RoboDK station: Robotska celija zadnja verzija.rdk

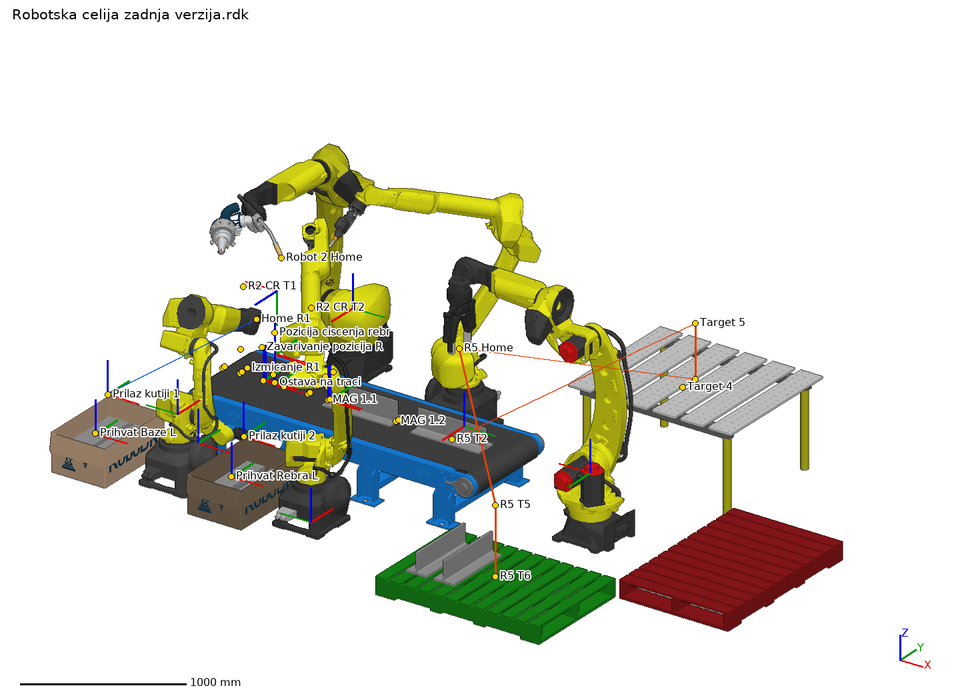
[picture v0: the station drawn from its stored meshes, robots at their saved joint values, targets as dots, program paths as lines]
Station Robotska celija zadnja verzija (saved by RoboDK 5.3.0). Poses are relative to the parent item; angles as X-Y-Z fixed-axis rotations.
  - program MAIN R12345 (8 instructions, listed below)
  - frame Frame Conveyor at (1000, 1000, 0) mm
    - robot Conveyor Belt Wide (2m): 1 axes
        modified DH rows (alpha deg, a mm, theta deg, d mm): 0, 0, 0, 0 linear
        base shift (0, 0, 0) mm, rotated rx 0 ry 90 rz 0 deg
        joint limits [-900000] to [900000]; home [0]; saved at [0]
  - frame R1 Frame at (1200, 500, 450) mm, rotated rx 0 ry 0 rz 90 deg
    - robot Fanuc M-10iD/16S: 6 axes
        modified DH rows (alpha deg, a mm, theta deg, d mm): 0, 0, 0, 450; -90, 75, -90, 0; 0, 440, 0, 0; -90, 195, 180, 555; 90, 0, 0, 0; -90, 0, 90, 90
        base shift (0, 0, -450) mm
        joint limits [-185, -90, -200, -190, -180, -450] to [185, 145, 200, 190, 180, 450]; home [0, 0, 0, 0, 0, 0]; saved at [0, 0, -25, 0, 0, 0]
      - tool OnRobot MG10 Magnetic Gripper, TCP at (0, 0, 93) mm, size 71 x 74.9 x 91.4 mm
  - object Kutija - baze at (500, 170, 0) mm, size 424.8 x 637.2 x 266.3 mm, geometry from Box-24x16in-Open.sld
    - object Baza L at (110, 310, 0) mm, rotated rx 0 ry 0 rz 90 deg, size 500 x 150 x 16 mm, geometry from Baza.step
      - object Baza at (0, 0, 16) mm, size 500 x 150 x 16 mm, geometry from Baza.step
        - object Baza at (0, 0, 16) mm, size 500 x 150 x 16 mm, geometry from Baza.step
          - object Baza at (0, 0, 16) mm, size 500 x 150 x 16 mm, geometry from Baza.step
            - object Baza at (0, 0, 16) mm, size 500 x 150 x 16 mm, geometry from Baza.step
              - object Baza at (0, 0, 16) mm, size 500 x 150 x 16 mm, geometry from Baza.step
    - object Baza D at (290, 310, 0) mm, rotated rx 0 ry 0 rz 90 deg, size 500 x 150 x 16 mm, geometry from Baza.step
      - object Baza at (0, 0, 16) mm, size 500 x 150 x 16 mm, geometry from Baza.step
        - object Baza at (0, 0, 16) mm, size 500 x 150 x 16 mm, geometry from Baza.step
          - object Baza at (0, 0, 16) mm, size 500 x 150 x 16 mm, geometry from Baza.step
            - object Baza at (0, 0, 16) mm, size 500 x 150 x 16 mm, geometry from Baza.step
              - object Baza at (0, 0, 16) mm, size 500 x 150 x 16 mm, geometry from Baza.step
                - object Baza at (0, 0, 16) mm, size 500 x 150 x 16 mm, geometry from Baza.step
                  - object Baza at (0, 0, 16) mm, size 500 x 150 x 16 mm, geometry from Baza.step
                    - object Baza at (0, 0, 16) mm, size 500 x 150 x 16 mm, geometry from Baza.step
                      - object Baza at (0, 0, 16) mm, size 500 x 150 x 16 mm, geometry from Baza.step
  - object Kutija - rebra at (1500, 170, 0) mm, size 424.8 x 637.2 x 266.3 mm, geometry from Box-24x16in-Open.sld
    - object Rebro L at (110, 310, 0) mm, rotated rx 0 ry 0 rz 90 deg, size 500 x 134 x 16 mm, geometry from Rebro.step
      - object Rebro at (0, 0, 16) mm, size 500 x 134 x 16 mm, geometry from Rebro.step
        - object Rebro at (0, 0, 16) mm, size 500 x 134 x 16 mm, geometry from Rebro.step
          - object Rebro at (0, 0, 16) mm, size 500 x 134 x 16 mm, geometry from Rebro.step
            - object Rebro at (0, 0, 16) mm, size 500 x 134 x 16 mm, geometry from Rebro.step
              - object Rebro at (0, 0, 16) mm, size 500 x 134 x 16 mm, geometry from Rebro.step
                - object Rebro at (0, 0, 16) mm, size 500 x 134 x 16 mm, geometry from Rebro.step
    - object Rebro D at (290, 310, 0) mm, rotated rx 0 ry 0 rz 90 deg, size 500 x 134 x 16 mm, geometry from Rebro.step
      - object Rebro at (0, 0, 16) mm, size 500 x 134 x 16 mm, geometry from Rebro.step
        - object Rebro at (0, 0, 16) mm, size 500 x 134 x 16 mm, geometry from Rebro.step
          - object Rebro at (0, 0, 16) mm, size 500 x 134 x 16 mm, geometry from Rebro.step
            - object Rebro at (0, 0, 16) mm, size 500 x 134 x 16 mm, geometry from Rebro.step
              - object Rebro at (0, 0, 16) mm, size 500 x 134 x 16 mm, geometry from Rebro.step
                - object Rebro at (0, 0, 16) mm, size 500 x 134 x 16 mm, geometry from Rebro.step
                  - object Rebro at (0, 0, 16) mm, size 500 x 134 x 16 mm, geometry from Rebro.step
                    - object Rebro at (0, 0, 16) mm, size 500 x 134 x 16 mm, geometry from Rebro.step
  - frame Prilaz Baza at (700, 480, 450) mm
    - target Home R1 (Cartesian target) at (500, 846.27, 304.84) mm, rotated rx 115 ry 0 rz -180 deg; joints [0, 0, -25, 0, 0, 0] of Fanuc M-10iD/16S
    - target Prilaz kutiji 1 (Cartesian target) at (0, 0, 0) mm, rotated rx 180 ry 0 rz -180 deg; joints [92.291, -14.525, -43.751, 180, -46.249, 87.709] of Fanuc M-10iD/16S
    - target Izmicanje R1 (Cartesian target) at (650, 537, 144.5) mm, rotated rx 0 ry -90 rz -90 deg; joints [-24.185, -35.816, -40.514, 34.657, -46.091, 244.385] of Fanuc M-10iD/16S
  - frame Baza L - prihvat at (610, 480, 160) mm
    - target Prihvat Baze L (Cartesian target) at (0, 0, 5) mm, rotated rx 180 ry 0 rz -180 deg; joints [91.941, 26.694, -76.673, 180, -13.327, -271.941] of Fanuc M-10iD/16S
  - frame Frame 5 at (1350, 1305, 366.5) mm
    - target Ostava na traci (Cartesian target) at (0, 0, 16) mm, rotated rx 180 ry 0 rz 90 deg; joints [169.445, -48.94, 177.796, 180, 92.204, -79.445] of Fanuc M-10iD/16S
    - target Ostava na traci Rebra (Cartesian target) at (0, -18, 78) mm, rotated rx 0 ry -90 rz -90 deg; joints [-13.947, 18.366, -65.349, 15.283, -66.122, 263.688] of Fanuc M-10iD/16S
    - target Target 3 (Cartesian target) at (400, -40.83, 183.83) mm, rotated rx -180 ry -45 rz 90 deg; joints [2.916, -45.786, -8.405, 0.478, -72.607, 356.977] of Fanuc ARC Mate 100iD/8L
    - target Target 4 (Cartesian target) at (2320, 965, 246.5) mm, rotated rx -180 ry 0 rz 90 deg; joints [-90, -0.762, -23.767, 0, -66.233, 0] of Fanuc M-20iD/35
    - target Target 5 (Cartesian target) at (2320, 1100, 623.5) mm, rotated rx -180 ry 0 rz 90 deg; joints [-90, 9.444, 0.734, 0, -90.734, 0] of Fanuc M-20iD/35
    - target Target 6 (Cartesian target) at (2320, 1100, 246.5) mm, rotated rx 180 ry 0 rz 90 deg; joints [-90, 8.37, -23.204, 0, -66.796, 0] of Fanuc M-20iD/35
  - program Prvi (4 instructions, listed below)
  - program Drugi (3 instructions, listed below)
  - program Treci (3 instructions, listed below)
  - program Cetvrti (3 instructions, listed below)
  - program PROGRAM 1 (6 instructions, listed below)
  - frame Prilaz Rebro at (1700, 480, 450) mm
    - target Prilaz kutiji 2 (Cartesian target) at (0, 0, 0) mm, rotated rx 180 ry 0 rz -180 deg; joints [87.709, -5.887, -173.705, 180, 83.705, 92.291] of Fanuc M-10iD/16S
  - frame Rebro L prihvat at (1610, 480, 154) mm
    - target Prihvat Rebra L (Cartesian target) at (0, 0, 0) mm, rotated rx 180 ry 0 rz -180 deg; joints [-92.793, 12.422, -85.191, 180, -4.809, 272.793] of Fanuc M-10iD/16S
    - target Target 2 (Cartesian target) at (0, 0, 0) mm, rotated rx 180 ry 0 rz -180 deg; joints [-92.793, 13.619, -86.144, 180, -3.856, 272.793] of Fanuc M-10iD/16S
    - target Target 3 (Cartesian target) at (0, 0, 0) mm, rotated rx 180 ry 0 rz -180 deg; joints [-92.793, 13.619, -86.144, 180, -3.856, 272.793] of Fanuc M-10iD/16S
    - target Target 4 (Cartesian target) at (0, 0, 0) mm, rotated rx 180 ry 0 rz -180 deg; joints [-92.793, 13.619, -86.144, 180, -3.856, 272.793] of Fanuc M-10iD/16S
    - target Target 5 (Cartesian target) at (0, 0, 0) mm, rotated rx 180 ry 0 rz -180 deg; joints [-92.793, 13.619, -86.144, 180, -3.856, 272.793] of Fanuc M-10iD/16S
    - target Target 6 (Cartesian target) at (0, 0, 0) mm, rotated rx 180 ry 0 rz -180 deg; joints [-92.793, 13.619, -86.144, 180, -3.856, 272.793] of Fanuc M-10iD/16S
    - target Target 7 (Cartesian target) at (0, 0, 0) mm, rotated rx 180 ry 0 rz -180 deg; joints [-92.793, 13.619, -86.144, 180, -3.856, 272.793] of Fanuc M-10iD/16S
    - target Target 8 (Cartesian target) at (0, 0, 0) mm, rotated rx 180 ry 0 rz -180 deg; joints [-92.793, 13.619, -86.144, 180, -3.856, 272.793] of Fanuc M-10iD/16S
    - target Target 9 (Cartesian target) at (0, 0, 0) mm, rotated rx 180 ry 0 rz -180 deg; joints [-92.793, 13.619, -86.144, 180, -3.856, 272.793] of Fanuc M-10iD/16S
    - target Target 10 (Cartesian target) at (0, 0, 0) mm, rotated rx 180 ry 0 rz -180 deg; joints [-92.793, 13.619, -86.144, 180, -3.856, 272.793] of Fanuc M-10iD/16S
  - frame Frame 8 at (1350, 1305, 566.5) mm
    - target Pozicija ciscenja rebra (Cartesian target) at (0, 0, 150) mm, rotated rx 0 ry 90 rz 90 deg; joints [-13.558, 0.356, -36.512, 22.063, -38.617, 432.428] of Fanuc M-10iD/16S
    - target Pozicija okrenute stranice 1 (Cartesian target) at (0.03, 0.03, 150.04) mm, rotated rx 89.99 ry 0 rz 180 deg; joints [-13.56, 0.36, -36.51, 22.06, -38.62, 342.43] of Fanuc M-10iD/16S
    - target Pozicija okrenute stranice 2 (Cartesian target) at (0.03, 0.03, 150.04) mm, rotated rx 0.43 ry -89.99 rz -90.44 deg; joints [-13.56, 0.36, -36.51, 22.06, -38.62, 252.43] of Fanuc M-10iD/16S
    - target Target 4 (Cartesian target) at (0, 0, 150) mm, rotated rx 0 ry 90 rz 90 deg; joints [-13.558, 0.356, -36.512, 22.063, -38.617, 432.428] of Fanuc M-10iD/16S
  - program Peti (3 instructions, listed below)
  - program Sesti (3 instructions, listed below)
  - program Sedmi (3 instructions, listed below)
  - program Osmi (3 instructions, listed below)
  - program Deveti (3 instructions, listed below)
  - program Deseti (3 instructions, listed below)
  - program PROGRAM 2 (11 instructions, listed below)
  - object Rebro at (1610, 480, 112) mm, rotated rx 0 ry 0 rz 90 deg, size 500 x 134 x 16 mm, geometry from Rebro.step
  - object Baza at (610, 480, 96) mm, rotated rx 0 ry 0 rz 90 deg, size 500 x 150 x 16 mm, geometry from Baza.step
  - object Baza at (610, 480.02, 128.03) mm, rotated rx 0 ry 0 rz -90 deg, size 500 x 150 x 16 mm, geometry from Baza.step
  - program Jedanaesti (3 instructions, listed below)
  - program Dvanaesti (5 instructions, listed below)
  - program Trinaesti (3 instructions, listed below)
  - program Robot 1 MAIN PROGRAM (4 instructions, listed below)
  - frame Fanuc ARC Mate 120iD/35 Base at (1300, 2200, 510) mm, rotated rx 0 ry 0 rz -90 deg
    - robot Fanuc ARC Mate 120iD/35: 6 axes
        modified DH rows (alpha deg, a mm, theta deg, d mm): 0, 0, 0, 425; -90, 75, -90, 0; 0, 840, 0, 0; -90, 215, 0, 890; 90, 0, 0, 0; -90, 0, 180, 90
        base shift (0, 0, -425) mm
        joint limits [-185, -130, -238, -200, -180, -450] to [185, 130, 220, 200, 180, 450]; home [0, 0, 0, 0, 0, 0]; saved at [0, 0, 0, 0, -15, 90]
      - tool OnRobot Dual Quick Tool Changer, TCP at (46.44, 0, 63.81) mm, rotated rx 0 ry 60 rz 0 deg, size 127 x 71 x 95.7 mm
      - tool Generic Laser Cutter, TCP at (-17.97, 0.01, 376.08) mm, rotated rx 178.57 ry -59.99 rz -178.26 deg, size 479.6 x 172.9 x 189.7 mm
      - tool Abicor Binzel 45deg Welding Gun, TCP at (-385.9, 0.01, 260.01) mm, rotated rx 173.72 ry -19.7 rz 130.69 deg, size 179.1 x 69.8 x 552.4 mm
    - target Zavarivanje pozicija R2 (Cartesian target) at (924.1, -25, 98.6) mm, rotated rx 60 ry 45 rz 180 deg; joints [5.612, -21.751, -19.966, 60.121, -83.046, -109.77] of Fanuc ARC Mate 120iD/35
    - target Robot 2 Home (Cartesian target) at (1303.08, 385.9, 964.39) mm, rotated rx -96.58 ry 50.97 rz 77.07 deg; joints [0, 0, 0, 0, -15, 90] of Fanuc ARC Mate 120iD/35
  - object Baza at (610, 480, 112) mm, rotated rx 0 ry 0 rz 90 deg, size 500 x 150 x 16 mm, geometry from Baza.step
  - Python program Pokretanje trake 1 (listed below)
  - Python program Pokretanje trake 2 (listed below)
  - frame Frame 18 at (1350, 1305, 577.5) mm
    - target R2 CB T1 (Cartesian target) at (250, 0, -40) mm, rotated rx 0 ry 90 rz 90 deg; joints [3.466, -49.475, -20.367, 92.478, -9.182, 214.863] of Fanuc ARC Mate 120iD/35
    - target R2 CB T2 (Cartesian target) at (-250, 0, -40) mm, rotated rx 0 ry 90 rz 90 deg; joints [-37.184, -31.629, -29.076, -101.453, -29.558, 65.206] of Fanuc ARC Mate 120iD/35
    - frame Frame 15 at (-75, -9.1, -198.9) mm
      - target ZAV1 T1 (Cartesian target) at (0, -1.73, 1.73) mm, rotated rx 60 ry 45 rz 90 deg; joints [5.725, -18.783, -33.331, 62.183, -76.662, 238.293] of Fanuc ARC Mate 120iD/35
      - target ZAV1 T2 (Cartesian target) at (-175, -1.73, 1.73) mm, rotated rx 60 ry 45 rz 90 deg; joints [-5.412, -18.825, -33.321, 67.05, -68.259, 242.481] of Fanuc ARC Mate 120iD/35
      - target ZAV1 T2.5 (Cartesian target) at (-300, -1.73, 1.73) mm, rotated rx 60 ry 45 rz 135 deg; joints [-16.96, -22.912, -32.182, 87.613, -22.309, 257.994] of Fanuc ARC Mate 120iD/35
      - target ZAV1 T4.75 (Cartesian target) at (385, 0, 70) mm, rotated rx 60 ry 45 rz 135 deg; joints [28.056, -18.642, -29.523, 69.642, -60.499, 250.402] of Fanuc ARC Mate 120iD/35
      - target ZAV1 T5 (Cartesian target) at (325, -1.73, 1.73) mm, rotated rx 60 ry 45 rz 90 deg; joints [24.816, -11.519, -34.828, 52.634, -89.199, 228.485] of Fanuc ARC Mate 120iD/35
      - target ZAV1 T6 (Cartesian target) at (150, -1.73, 1.73) mm, rotated rx 60 ry 45 rz 90 deg; joints [14.971, -16.455, -33.885, 57.833, -83.056, 233.9] of Fanuc ARC Mate 120iD/35
    - frame Frame 16 at (-75, 9.1, -198.9) mm
      - target ZAV1 T2.75 (Cartesian target) at (-300, 1.73, 1.73) mm, rotated rx 60 ry 45 rz -135 deg; joints [-27.007, -18.272, -33.459, 109.336, 61.454, 293.444] of Fanuc ARC Mate 120iD/35
      - target ZAV1 T3 (Cartesian target) at (-175, 1.73, 1.73) mm, rotated rx 60 ry 45 rz -90 deg; joints [-19.437, -14.977, -34.201, 126.554, 88.605, 308.95] of Fanuc ARC Mate 120iD/35
      - target ZAV1 T4 (Cartesian target) at (325, 1.73, 1.73) mm, rotated rx 60 ry 45 rz -90 deg; joints [11.711, -17.948, -33.538, 111.866, 66.329, 295.578] of Fanuc ARC Mate 120iD/35
      - target ZAV1 T4.5 (Cartesian target) at (385, 0, 70) mm, rotated rx 60 ry 45 rz -135 deg; joints [18.599, -24.807, -27.778, 102.936, 24.85, 270.405] of Fanuc ARC Mate 120iD/35
  - frame Frame 19 at (1350, 1331, 983.5) mm, rotated rx -90 ry 0 rz -180 deg
    - target R2 CR T1 (Cartesian target) at (250, 40, 0) mm, rotated rx -180 ry 0 rz 90 deg; joints [-38.392, -35.898, -5.358, 117.561, 34.365, -159.672] of Fanuc ARC Mate 120iD/35
    - target R2 CR T2 (Cartesian target) at (-250, 40, 0) mm, rotated rx -180 ry 0 rz 90 deg; joints [3.619, -49.197, 1.409, 24.228, -23.239, 284.855] of Fanuc ARC Mate 120iD/35
  - program Robot 2 - ciscenje baze (3 instructions, listed below)
  - program Prog26 (3 instructions, listed below)
  - program Prog27 (3 instructions, listed below)
  - program Prog28 (3 instructions, listed below)
  - program Prog29 (3 instructions, listed below)
  - program Prog30 (3 instructions, listed below)
  - program Robot 2 - ciscenje rebra (5 instructions, listed below)
  - program Prog32A (3 instructions, listed below)
  - program Prog33A (3 instructions, listed below)
  - program Prog34A (3 instructions, listed below)
  - program Prog35A (3 instructions, listed below)
  - program Prog36A (3 instructions, listed below)
  - program Prog37A (3 instructions, listed below)
  - program Prog38A (3 instructions, listed below)
  - program Prog39A (3 instructions, listed below)
  - program Prog40A (3 instructions, listed below)
  - program Prog41A (3 instructions, listed below)
  - program Prog42A (3 instructions, listed below)
  - program Prog43A (3 instructions, listed below)
  - program Prog44A (3 instructions, listed below)
  - program Robot 2 - korijenski zavar (17 instructions, listed below)
  - program Robot 2 MAIN PROGRAM (6 instructions, listed below)
  - frame Fanuc ARC Mate 100iD/8L Base 1 at (2180, 500, 0) mm, rotated rx 0 ry 0 rz 90 deg
    - robot Fanuc ARC Mate 100iD/8L: 6 axes
        modified DH rows (alpha deg, a mm, theta deg, d mm): 0, 0, 0, 0; -90, 75, -90, 0; 0, 840, 0, 0; -90, 195, 0, 1100; 90, 0, 0, 0; -90, 0, 180, 75
        base shift (0, 0, 450) mm
        joint limits [-185, -100, -185, -190, -180, -450] to [185, 160, 275, 190, 180, 450]; home [0, 0, 0, 0, 0, 0]; saved at [35.77, -32.548, -15.249, 5.679, -67.528, 322.389]
      - tool Fronius MTB500i Welding Gun, TCP at (86, 0, 451.5) mm, rotated rx 0 ry 36 rz 0 deg, size 139 x 105 x 455.9 mm
    - frame MAG zavarivanje naprijed at (797, 430, 377.5) mm, rotated rx 0 ry 0 rz -90 deg
      - target MAG 1.0 (Cartesian target) at (0, -32.83, 172.83) mm, rotated rx -180 ry -45 rz 90 deg; joints [35.77, -32.548, -15.249, 5.679, -67.528, 322.389] of Fanuc ARC Mate 100iD/8L
      - target MAG 1.1 (Cartesian target) at (0, -2.83, 2.83) mm, rotated rx 180 ry -45 rz 90 deg; joints [34.448, -27.568, -26.042, 6.08, -56.665, 322.532] of Fanuc ARC Mate 100iD/8L
      - target MAG 1.2 (Cartesian target) at (500, -2.83, 2.83) mm, rotated rx 180 ry -45 rz 90 deg; joints [-6.372, -40.231, -20.595, -181.143, 60.464, -173.143] of Fanuc ARC Mate 100iD/8L
  - program R3 P1 (3 instructions, listed below)
  - program R3 P2 (3 instructions, listed below)
  - program R3 P3 (3 instructions, listed below)
  - program Robot 3 MAIN PROGRAM (7 instructions, listed below)
  - frame Fanuc ARC Mate 100iD/8L Base 2 at (2180, 2110, 0) mm, rotated rx 0 ry 0 rz -90 deg
    - robot Fanuc ARC Mate 100iD/8L: 6 axes
        modified DH rows (alpha deg, a mm, theta deg, d mm): 0, 0, 0, 0; -90, 75, -90, 0; 0, 840, 0, 0; -90, 195, 0, 1100; 90, 0, 0, 0; -90, 0, 180, 75
        base shift (0, 0, 450) mm
        joint limits [-185, -100, -185, -190, -180, -450] to [185, 160, 275, 190, 180, 450]; home [0, 0, 0, 0, 0, 0]; saved at [-35.77, -32.548, -15.249, -185.679, 67.528, 217.611]
      - tool Fronius MTB500i Welding Gun, TCP at (86, 0, 451.5) mm, rotated rx 0 ry 36 rz 0 deg, size 139 x 105 x 455.9 mm
    - frame MAG Zavarivanje nazad at (797, -430, 377.5) mm, rotated rx 0 ry 0 rz 90 deg
      - target MAG 2.0 (Cartesian target) at (0, 32.83, 172.83) mm, rotated rx 180 ry -45 rz -90 deg; joints [-35.77, -32.548, -15.249, -185.679, 67.528, 217.611] of Fanuc ARC Mate 100iD/8L
      - target MAG 2.1 (Cartesian target) at (0, 2.83, 2.83) mm, rotated rx 180 ry -45 rz -90 deg; joints [-34.448, -27.568, -26.042, -6.08, -56.665, 37.468] of Fanuc ARC Mate 100iD/8L
      - target MAG 2.2 (Cartesian target) at (500, 2.83, 2.83) mm, rotated rx 180 ry -45 rz -90 deg; joints [6.372, -40.231, -20.595, 1.143, -60.464, -6.857] of Fanuc ARC Mate 100iD/8L
  - program R4 P1 (3 instructions, listed below)
  - program R4 P2 (3 instructions, listed below)
  - program R4 P3 (3 instructions, listed below)
  - program Robot 4 MAIN PROGRAM (6 instructions, listed below)
  - object Pallet 1200x800mm at (4270, -95, 130) mm, rotated rx 0 ry 0 rz 90 deg, size 800 x 1200 x 125 mm, geometry from Pallet-1200x800mm.sld
  - frame Fanuc M-20iD/35 Base at (3670, 1305, 425) mm, rotated rx 0 ry 0 rz 180 deg
    - robot Fanuc M-20iD/35: 6 axes
        modified DH rows (alpha deg, a mm, theta deg, d mm): 0, 0, 0, 425; -90, 75, -90, 0; 0, 840, 0, 0; -90, 215, 0, 890; 90, 0, 0, 0; -90, 0, 0, 90
        base shift (0, 0, -425) mm
        joint limits [-170, -100, -200, -200, -180, -450] to [170, 160, 200, 200, 180, 450]; home [0, 0, 0, 0, 0, 0]; saved at [0, 0, 0, 0, -90, -90]
      - tool RobotiQ 2F-140 Gripper (Open), TCP at (0, 0, 400) mm, size 278.1 x 150 x 407.5 mm
    - target R5 Home (Cartesian target) at (965, 0, 565) mm, rotated rx -180 ry 0 rz -90 deg; joints [0, 0, 0, 0, -90, -90] of Fanuc M-20iD/35
    - target R5 T2 (Cartesian target) at (1020, 0, -60.5) mm, rotated rx 180 ry 0 rz -90 deg; joints [0, 8.362, -39.595, 0, -50.405, -90] of Fanuc M-20iD/35
    - target R5 T3 (Cartesian target) at (0, -1100, 565) mm, rotated rx -180 ry 0 rz -90 deg; joints [-90, 9.444, 0.734, 0, -90.734, 0] of Fanuc M-20iD/35
    - target R5 T4 (Cartesian target) at (0, -1100, 188) mm, rotated rx -180 ry 0 rz -90 deg; joints [-90, 8.37, -23.204, 0, -66.796, 0] of Fanuc M-20iD/35
    - target R5 T5 (Cartesian target) at (0, 1000, 185) mm, rotated rx -180 ry 0 rz 0 deg; joints [90, 1.659, -23.94, 0, -66.06, -90] of Fanuc M-20iD/35
    - target R5 T6 (Cartesian target) at (0, 1000, -292) mm, rotated rx -180 ry 0 rz 0 deg; joints [90, 16.574, -55.115, 0, -34.885, -90] of Fanuc M-20iD/35
  - program Robot 5 MAIN PROGRAM (18 instructions, listed below)
  - object Table 1200x1000mm (Welding) at (3670, 2405, 610) mm, rotated rx 0 ry 0 rz -180 deg, size 1193.8 x 965.2 x 609.6 mm, geometry from Table-1200x1000mm-Welding.sld
  - object Pallet 1200x800mm at (5100, 1905, 130) mm, rotated rx 0 ry 0 rz 180 deg, size 800 x 1200 x 125 mm, geometry from Pallet-1200x800mm.sld
  - object Baza na traci 1 at (2000, 1305, 361.5) mm, size 500 x 150 x 16 mm, geometry from Baza.step
  - object Rebro na podlozi 1 at (2000, 1313, 444.5) mm, rotated rx 90 ry 0 rz 0 deg, size 500 x 134 x 16 mm, geometry from Rebro.step
  - object Baza na traci 2 at (610, 480, 144) mm, rotated rx 0 ry 0 rz 90 deg, size 500 x 150 x 16 mm, geometry from Baza.step
  - object Rebro na podlozi 2 at (1610, 480, 128) mm, rotated rx 0 ry 0 rz 90 deg, size 500 x 134 x 16 mm, geometry from Rebro.step
  - object T_profil 2 at (3465, 55, 130) mm, size 150 x 500 x 150 mm, geometry from T_profil.step
    - object T_profil 1 at (-200, 0, 0) mm, size 150 x 500 x 150 mm, geometry from T_profil.step
  - object T_profil na traci at (2900, 1305, 361.5) mm, rotated rx 0 ry 0 rz 90 deg, size 150 x 500 x 150 mm, geometry from T_profil.step
  - object T_profil at (2250, 1305, 361.5) mm, rotated rx 0 ry 0 rz 90 deg, size 150 x 500 x 150 mm, geometry from T_profil.step
  - Python program Sakrij/pokazi (listed below)
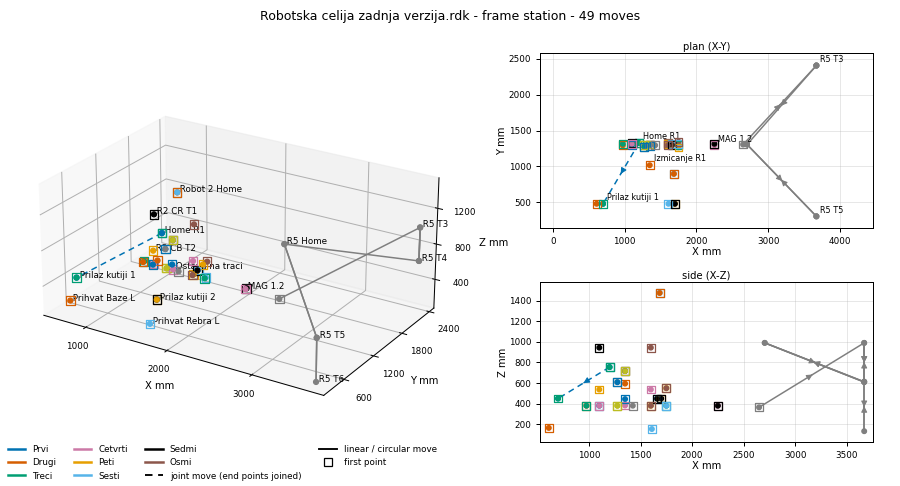
[picture p0: tool path of Robotska celija zadnja verzija.rdk in frame station, 49 of 49 moves have a stored position in this frame; points joined in program order, loops and branches not executed]

--- program MAIN R12345 (robot Fanuc M-10iD/16S) ---
  Run Robot 1 MAIN PROGRAM
  Run Robot 2 MAIN PROGRAM
  Run Robot 3 MAIN PROGRAM
  Run Robot 4 MAIN PROGRAM
  Run Robot 5 MAIN PROGRAM
  Pause 73.0 s
  Run Pokretanje trake 1
  Run Pokretanje trake 2

--- program Prvi (robot Fanuc M-10iD/16S) ---
  Set Ref.: Prilaz Baza
  Set Tool: OnRobot MG10 Magnetic Gripper
  MoveJ (Home) -> target Home R1
  MoveJ (Prilaz kutiji 1)

--- program Drugi (robot Fanuc M-10iD/16S) ---
  Set Ref.: Baza L - prihvat
  Set Tool: OnRobot MG10 Magnetic Gripper
  MoveL (Prihvat Baze L)

--- program Treci (robot Fanuc M-10iD/16S) ---
  Set Ref.: Prilaz Baza
  Set Tool: OnRobot MG10 Magnetic Gripper
  MoveL (Prilaz kutiji 1)

--- program Cetvrti (robot Fanuc M-10iD/16S) ---
  Set Ref.: Frame 5
  Set Tool: OnRobot MG10 Magnetic Gripper
  MoveL (Ostava na traci)

--- program PROGRAM 1 (robot Fanuc M-10iD/16S) ---
  Call Prvi
  Call Drugi
  Attach to OnRobot MG10 Magnetic Gripper
  Call Treci
  Call Cetvrti
  Detach from OnRobot MG10 Magnetic Gripper

--- program Peti (robot Fanuc M-10iD/16S) ---
  Set Ref.: Prilaz Rebro
  Set Tool: OnRobot MG10 Magnetic Gripper
  MoveL (Prilaz kutiji 2)

--- program Sesti (robot Fanuc M-10iD/16S) ---
  Set Ref.: Rebro L prihvat
  Set Tool: OnRobot MG10 Magnetic Gripper
  MoveL (Prihvat Rebra L)

--- program Sedmi (robot Fanuc M-10iD/16S) ---
  Set Ref.: Prilaz Rebro
  Set Tool: OnRobot MG10 Magnetic Gripper
  MoveL (Prilaz kutiji 2)

--- program Osmi (robot Fanuc M-10iD/16S) ---
  Set Ref.: Frame 8
  Set Tool: OnRobot MG10 Magnetic Gripper
  MoveL (Pozicija ciscenja rebra)

--- program Deveti (robot Fanuc M-10iD/16S) ---
  Set Ref.: Frame 8
  Set Tool: OnRobot MG10 Magnetic Gripper
  MoveJ (Pozicija okrenute stranice 1)

--- program Deseti (robot Fanuc M-10iD/16S) ---
  Set Ref.: Frame 8
  Set Tool: OnRobot MG10 Magnetic Gripper
  MoveJ (Pozicija okrenute stranice 2)

--- program PROGRAM 2 (robot Fanuc M-10iD/16S) ---
  Call Peti
  Call Sesti
  Attach to OnRobot MG10 Magnetic Gripper
  Call Sedmi
  Call Osmi
  Pause 3.5 s
  Call Deveti
  Call Deseti
  Call Jedanaesti
  Pause 38.0 s
  Detach from OnRobot MG10 Magnetic Gripper

--- program Jedanaesti (robot Fanuc M-10iD/16S) ---
  Set Ref.: Frame 5
  Set Tool: OnRobot MG10 Magnetic Gripper
  MoveL (Ostava na traci Rebra)

--- program Dvanaesti (robot Fanuc M-10iD/16S) ---
  Set Ref.: Prilaz Baza
  Set Tool: OnRobot MG10 Magnetic Gripper
  MoveL (Izmicanje R1)
  Pause 7.0 s
  Run Trinaesti

--- program Trinaesti (robot Fanuc M-10iD/16S) ---
  Set Ref.: Prilaz Baza
  Set Tool: OnRobot MG10 Magnetic Gripper
  MoveJ (Home) -> target Home R1

--- program Robot 1 MAIN PROGRAM (robot Fanuc M-10iD/16S) ---
  Set speed (800.0 mm/s)
  Call PROGRAM 1
  Call PROGRAM 2
  Call Dvanaesti

--- Python program Pokretanje trake 1 ---
import time
from robolink import *
from robodk import *

RDK = Robolink()

t_profil = RDK.Item('T_profil')

t_profil_postoji = t_profil.Valid()

if t_profil_postoji:
    t_profil_pocetna = t_profil.Pose()
else:
    print("Upozorenje: Objekt 'T_profil' nije pronađen.")

trajanje_sekundi = 2.0
ukupni_pomak = 650.0

# Promjenom parametra trajanje_sekundi mijenja se vrijeme pomicanja po traci
# Promjenom parametra ukupni_pomak mijenja se duljina pomicanja po traci

RDK.Render(False)

pocetno_vrijeme = time.time()
proteklo_vrijeme = 0.0

while proteklo_vrijeme < trajanje_sekundi:
    proteklo_vrijeme = time.time() - pocetno_vrijeme

    udio = min(proteklo_vrijeme / trajanje_sekundi, 1.0)

    trenutni_pomak = transl(ukupni_pomak * udio, 0, 0)

    if t_profil_postoji:
        t_profil.setPose(trenutni_pomak * t_profil_pocetna)

    RDK.Render()

    time.sleep(0.01)

RDK.Render(True)

# Pozivom programa se T profil pomiče trakom (simulira se mehanizam trake)

--- Python program Pokretanje trake 2 ---
import time
from robolink import *
from robodk import *

RDK = Robolink()

baza = RDK.Item('Baza na traci 2')
rebro = RDK.Item('Rebro na podlozi 2')

baza_postoji = baza.Valid()
rebro_postoji = rebro.Valid()

if baza_postoji:
    baza_pocetna = baza.Pose()
if rebro_postoji:
    rebro_pocetna = rebro.Pose()

trajanje_sekundi = 2.0
ukupni_pomak = 650.0

# Promjenom parametra trajanje_sekundi mijenja se vrijeme pomicanja po traci
# Promjenom parametra ukupni_pomak mijenja se duljina pomicanja po traci

RDK.Render(False)

pocetno_vrijeme = time.time()
proteklo_vrijeme = 0.0

while proteklo_vrijeme < trajanje_sekundi:
    proteklo_vrijeme = time.time() - pocetno_vrijeme

    udio = min(proteklo_vrijeme / trajanje_sekundi, 1.0)

    trenutni_pomak = transl(ukupni_pomak * udio, 0, 0)

    if baza_postoji:
        baza.setPose(trenutni_pomak * baza_pocetna)
    if rebro_postoji:
        rebro.setPose(trenutni_pomak * rebro_pocetna)

    RDK.Render()

    time.sleep(0.01)

RDK.Render(True)

# Pozivom programa se T profil pomiče trakom (simulira se mehanizam trake)

--- program Robot 2 - ciscenje baze (robot Fanuc ARC Mate 120iD/35) ---
  Call Prog26
  Call Prog27
  Call Prog28

--- program Prog26 (robot Fanuc ARC Mate 120iD/35) ---
  Set Ref.: Frame 18
  Set Tool: Generic Laser Cutter
  MoveL (R2 CB T1)

--- program Prog27 (robot Fanuc ARC Mate 120iD/35) ---
  Set Ref.: Frame 18
  Set Tool: Generic Laser Cutter
  MoveL (R2 CB T2)

--- program Prog28 (robot Fanuc ARC Mate 120iD/35) ---
  Set Ref.: Fanuc ARC Mate 120iD/35 Base
  Set Tool: Generic Laser Cutter
  MoveL (Robot 2 Home)

--- program Prog29 (robot Fanuc ARC Mate 120iD/35) ---
  Set Ref.: Frame 19
  Set Tool: Generic Laser Cutter
  MoveL (Target 1) -> target R2 CR T1

--- program Prog30 (robot Fanuc ARC Mate 120iD/35) ---
  Set Ref.: Frame 19
  Set Tool: Generic Laser Cutter
  MoveL (Target 2) -> target R2 CR T2

--- program Robot 2 - ciscenje rebra (robot Fanuc ARC Mate 120iD/35) ---
  Call Prog29
  Call Prog30
  Call Prog28
  Pause 1.5 s
  Call Prog32A

--- program Prog32A (robot Fanuc ARC Mate 120iD/35) ---
  Set Ref.: R2 Frame -> Fanuc ARC Mate 120iD/35 Base
  Set Tool: Abicor Binzel 45deg Welding Gun
  MoveL (Home2 R2) -> target Zavarivanje pozicija R2

--- program Prog33A (robot Fanuc ARC Mate 120iD/35) ---
  Set Ref.: Frame 15
  Set Tool: Abicor Binzel 45deg Welding Gun
  MoveL (ZAV1 T1)

--- program Prog34A (robot Fanuc ARC Mate 120iD/35) ---
  Set Ref.: Frame 15
  Set Tool: Abicor Binzel 45deg Welding Gun
  MoveL (ZAV1 T2)

--- program Prog35A (robot Fanuc ARC Mate 120iD/35) ---
  Set Ref.: Frame 15
  Set Tool: Abicor Binzel 45deg Welding Gun
  MoveL (ZAV1 T2.5)

--- program Prog36A (robot Fanuc ARC Mate 120iD/35) ---
  Set Ref.: Frame 16
  Set Tool: Abicor Binzel 45deg Welding Gun
  MoveJ (ZAV1 T2.75)

--- program Prog37A (robot Fanuc ARC Mate 120iD/35) ---
  Set Ref.: Frame 16
  Set Tool: Abicor Binzel 45deg Welding Gun
  MoveL (ZAV1 T3)

--- program Prog38A (robot Fanuc ARC Mate 120iD/35) ---
  Set Ref.: Frame 16
  Set Tool: Abicor Binzel 45deg Welding Gun
  MoveL (ZAV1 T4)

--- program Prog39A (robot Fanuc ARC Mate 120iD/35) ---
  Set Ref.: Frame 16
  Set Tool: Abicor Binzel 45deg Welding Gun
  MoveL (ZAV1 T4.5)

--- program Prog40A (robot Fanuc ARC Mate 120iD/35) ---
  Set Ref.: Frame 15
  Set Tool: Abicor Binzel 45deg Welding Gun
  MoveL (ZAV1 T4.75)

--- program Prog41A (robot Fanuc ARC Mate 120iD/35) ---
  Set Ref.: Frame 15
  Set Tool: Abicor Binzel 45deg Welding Gun
  MoveL (ZAV1 T5)

--- program Prog42A (robot Fanuc ARC Mate 120iD/35) ---
  Set Ref.: Frame 15
  Set Tool: Abicor Binzel 45deg Welding Gun
  MoveL (ZAV1 T6)

--- program Prog43A (robot Fanuc ARC Mate 120iD/35) ---
  Set Ref.: Frame 15
  Set Tool: Abicor Binzel 45deg Welding Gun
  MoveL (ZAV1 T1)

--- program Prog44A (robot Fanuc ARC Mate 120iD/35) ---
  Set Ref.: R2 Frame -> Fanuc ARC Mate 120iD/35 Base
  Set Tool: Abicor Binzel 45deg Welding Gun
  MoveL (Home2 R2) -> target Zavarivanje pozicija R2

--- program Robot 2 - korijenski zavar (robot Fanuc ARC Mate 120iD/35) ---
  Call Prog33A
  Set speed (26.0 mm/s)
  Call Prog34A
  Set speed (800.0 mm/s)
  Call Prog35A
  Call Prog36A
  Call Prog37A
  Set speed (26.0 mm/s)
  Call Prog38A
  Set speed (800.0 mm/s)
  Call Prog39A
  Call Prog40A
  Call Prog41A
  Set speed (26.0 mm/s)
  Call Prog43A
  Set speed (800.0 mm/s)
  Call Prog44A

--- program Robot 2 MAIN PROGRAM (robot Fanuc ARC Mate 120iD/35) ---
  Set speed (800.0 mm/s)
  Pause 7.0 s
  Call Robot 2 - ciscenje baze
  Call Robot 2 - ciscenje rebra
  Call Robot 2 - korijenski za...: Robot 2 - korijenski zavar
  MoveL (Robot 2 Home)

--- program R3 P1 (robot Fanuc ARC Mate 100iD/8L) ---
  Set Ref.: MAG zavarivanje naprijed
  Set Tool: Fronius MTB500i Welding Gun
  MoveJ (MAG 1.1)

--- program R3 P2 (robot Fanuc ARC Mate 100iD/8L) ---
  Set Ref.: MAG zavarivanje naprijed
  Set Tool: Fronius MTB500i Welding Gun
  MoveL (MAG 1.2)

--- program R3 P3 (robot Fanuc ARC Mate 100iD/8L) ---
  Set Ref.: MAG zavarivanje naprijed
  Set Tool: Fronius MTB500i Welding Gun
  MoveL (MAG 1.0)

--- program Robot 3 MAIN PROGRAM (robot Fanuc ARC Mate 100iD/8L) ---
  Set speed (1000.0 mm/s)
  Call R3 P1
  Set speed (7.2 mm/s)
  Call R3 P2
  Set speed (1000.0 mm/s)
  Call R3 P3
  Call Sakrij/pokazi

--- program R4 P1 (robot Fanuc ARC Mate 100iD/8L) ---
  Set Ref.: MAG Zavarivanje nazad
  Set Tool: Fronius MTB500i Welding Gun
  MoveL (MAG 2.1)

--- program R4 P2 (robot Fanuc ARC Mate 100iD/8L) ---
  Set Ref.: MAG Zavarivanje nazad
  Set Tool: Fronius MTB500i Welding Gun
  MoveL (MAG 2.2)

--- program R4 P3 (robot Fanuc ARC Mate 100iD/8L) ---
  Set Ref.: MAG Zavarivanje nazad
  Set Tool: Fronius MTB500i Welding Gun
  MoveL (MAG 2.0)

--- program Robot 4 MAIN PROGRAM (robot Fanuc ARC Mate 100iD/8L) ---
  Set speed (1000.0 mm/s)
  Call R4 P1
  Set speed (7.2 mm/s)
  Call R4 P2
  Set speed (1000.0 mm/s)
  Call R4 P3

--- program Robot 5 MAIN PROGRAM (robot Fanuc M-20iD/35) ---
  Set speed (700.0 mm/s)
  Set Ref.: Fanuc M-20iD/35 Base
  Set Tool: RobotiQ 2F-140 Gripper (Open)
  MoveL (R5 T2)
  Attach to RobotiQ 2F-140 Gripper (Open)
  MoveL (R5 T3)
  MoveL (R5 T4)
  Detach from RobotiQ 2F-140 Gripper (Open)
  MoveL (R5 T3)
  Pause 52.9 s
  MoveL (R5 T4)
  Attach to RobotiQ 2F-140 Gripper (Open)
  MoveL (R5 Home)
  MoveL (R5 T5)
  MoveL (R5 T6)
  Detach from RobotiQ 2F-140 Gripper (Open)
  MoveL (R5 T5)
  MoveL (R5 Home)

--- Python program Sakrij/pokazi ---
from robolink import *
from robodk import *

RDK = Robolink()

baza = RDK.Item("Baza na traci 1")
rebro = RDK.Item("Rebro na podlozi 1")
t_profil = RDK.Item("T_profil")

if t_profil.Valid():
    t_profil.setVisible(True)

if baza.Valid():
    baza.setVisible(False)

if rebro.Valid():
    rebro.setVisible(False)

# Pozivanjem programa T profil postaje vidljiv, a baza i rebro
# koji se nalaze na njegovom mjestu postaju nevidljivi.
